// TIA Portal V17 export
// export: Created 2022-07-20T07:01:32.0836493Z, ExportSetting WithDefaults, DisplayName Totally Integrated Automation Portal, DisplayVersion V17, DisplayName TIA Portal Openness, DisplayVersion V17, DisplayName TIA Portal Version Control Interface, DisplayVersion V17, DisplayName SINAMICS Startdrive Advanced, DisplayVersion V17, DisplayName SINAMICS Startdrive G130, G150, S120, S150, SINAMICS MV, S210, DisplayVersion V17, DisplayName SINAMICS Startdrive G110M, G120, G120C, G120D, G120P, G115D, DisplayVersion V17, DisplayName STEP 7 Professional, DisplayVersion V17, DisplayName STEP 7 Safety, DisplayVersion V17, DisplayName WinCC Advanced, DisplayVersion V17
FUNCTION_BLOCK "FB10341_Bladder"   // FB10341, LAD
TITLE = FB10341_Bladder
{ S7_Optimized_Access := 'TRUE' }
VERSION : 0.1
// stored: AutoNumber false, IsIECCheckEnabled false, IsRetainMemResEnabled false, MemoryReserve 100, SetENOAutomatically false, UDAEnableTagReadback false
   VAR_INPUT
      RequestAcknowledge : Bool;
   END_VAR
   VAR_OUTPUT
      ActiveBladder : Bool;
      BladderActivated : Bool;
      BladderInError : Bool;
   END_VAR
   VAR_IN_OUT
      RequestActiveBladder : Bool;
   END_VAR
   VAR
      R_TRIG_RequestActiveBladder : R_TRIG;
      F_TRIG_RequestActiveBladder { S7_SetPoint := 'True'} : F_TRIG;
      TON_BladderActivated { S7_SetPoint := 'True'} : TON_TIME;
      TON_BladderNotActivated { S7_SetPoint := 'True'} : TON_TIME;
      TON_BladderInError { S7_SetPoint := 'True'} : TON_TIME;
   END_VAR
BEGIN

REGION Network 1 (SCL): First Scan
   IF "FirstScan" THEN
       #ActiveBladder := FALSE;
       #BladderActivated := FALSE;
   END_IF;
END_REGION

REGION Network 2 (SCL): Edge Signals & Timers
   REGION EDGE SIGNALS
       #R_TRIG_RequestActiveBladder(CLK := #RequestActiveBladder);

       #F_TRIG_RequestActiveBladder(CLK := #RequestActiveBladder);
   END_REGION

   REGION TIMERS
       #TON_BladderActivated(IN := #ActiveBladder,
                             PT := T#1s);
       #TON_BladderNotActivated(IN := NOT (#ActiveBladder),
                                PT := T#1s);
       #TON_BladderInError(IN := #RequestActiveBladder AND NOT(#ActiveBladder)
                           OR #RequestActiveBladder  AND NOT(#BladderActivated)
                           OR NOT(#RequestActiveBladder) AND #ActiveBladder
                           OR NOT(#RequestActiveBladder) AND #BladderActivated, PT := T#10s);
   END_REGION
END_REGION

REGION Network 3 (SCL): Bladder Management
   IF #R_TRIG_RequestActiveBladder.Q THEN
       #ActiveBladder := TRUE;
   ELSIF #F_TRIG_RequestActiveBladder.Q THEN
       #ActiveBladder := FALSE;
   END_IF;
END_REGION

REGION Network 4 (SCL): States
   IF #TON_BladderActivated.Q THEN
       #BladderActivated := TRUE;
   ELSIF #TON_BladderNotActivated.Q THEN
       #BladderActivated := FALSE;
   END_IF;

   IF #TON_BladderInError.Q THEN
       #BladderInError := TRUE;
   ELSIF #RequestAcknowledge THEN
       #BladderInError := FALSE;
   END_IF;
END_REGION
END_FUNCTION_BLOCK
